(* CODESYS project codesys_git_test

Project tree, tasks and I/O mapping:
  Device : CODESYS Control for PFC200 SL, 3S - Smart Software Solutions GmbH, version 4.1.0.0
    application Application
      libraries: Standard, * (System)
      task MainTask (cyclic, interval t#20ms, priority 1) calls PLC_PRG
      program PLC_PRG [ST]
    Pfc200Bus : Wago PFC200 internal bus, 3S - Smart Software Solutions GmbH, version 4.1.0.0
*)

// Device/Application/PLC_PRG
PROGRAM PLC_PRG
VAR
	iMyNum	: INT;
END_VAR

iMyNum := iMyNum + 1;

END_PROGRAM
